# EPICS substitutions: adsApp/Db/FB_DriveVirtual.substitutions
#
#    This file is part of epics-twincat-ads.
#
#    epics-twincat-ads is free software: you can redistribute it and/or modify it under the terms of the GNU Lesser General Public License as published by the Free Software Foundation, either version 3 of the License, or (at your option) any later version.
#
#    epics-twincat-ads is distributed in the hope that it will be useful, but WITHOUT ANY WARRANTY; without even the implied warranty of MERCHANTABILITY or FITNESS FOR A PARTICULAR PURPOSE. See the GNU Lesser General Public License for more details.
#
#    You should have received a copy of the GNU Lesser General Public License along with epics-twincat-ads. If not, see <https://www.gnu.org/licenses/>.
#
file "FB_DriveVirtual_v1_01.template"
{
pattern
{P,      PORT,      A, P, VP,     VI, VN   }
{ADSTEST:,  ADS_1,  "", "" , Main.M, 1, "" }
}
